DATA_BLOCK "dbVizu"
{ S7_Optimized_Access := 'FALSE' }
VERSION : 0.1
NON_RETAIN
   STRUCT
      iSecond : Int;
      iWMU_Temp : Int;   // 0,1°C
      iWMU_Ticks : Int;   // dílky   #0.1#°C#
      diAH1_Weight : DInt;   // 1g
      diAK1_Weight : DInt;   // 1g
      diAK2_Weight : DInt;   // 1g
      iAH1_TempSide : Int;   // 0,1°C
      iAH1_TempBottom : Int;   // 0,1°C
      iAK1_TempSide : Int;   // 0,1°C
      iAK1_TempBottom : Int;   // 0,1°C
      iAK2_TempSide : Int;   // 0,1°C
      iAK2_TempBottom : Int;   // 0,1°C
      iPIG1_Pressure : Int;   // 0,01 Bar
      iAK1_Pressure : Int;   // 0,01 Bar
      iAK2_Pressure : Int;   // 0,01 Bar
      iAH1_RCP_No : Int;   // cislo RCP
      usiAH1_RCP_Status : Byte;   // stav
      usiAH1_RCP_Step : Byte;   // krok
      sAH1_RCP_Name : String[40];   // jmeno RCP
      diAH1_RCP_TotalAmount : DInt;   // 0,001 kg
      iAH1_RCP_Shower_Step : Int;
      iAH1_RCP_TA : Int;
      diAH1_RCP_Mixture_need : DInt;   // 0,001 kg
      diAH1_RCP_Mixture_done : DInt;   // 0,001 kg
      diAH1_RCP_Mixing1_need : DInt;   // 0,016666667 min
      diAH1_RCP_Mixing1_done : DInt;   // 0,016666667 min
      diAH1_RCP_ManComp1_need : DInt;   // 0,001 kg
      diAH1_RCP_ManComp1_done : DInt;   // 0,001 kg
      diAH1_RCP_Mixing2_need : DInt;   // 0,016666667 min
      diAH1_RCP_Mixing2_done : DInt;   // 0,016666667 min
      diAH1_RCP_AutComp1_need : DInt;   // 0,001 kg
      diAH1_RCP_AutComp1_done : DInt;   // 0,001 kg
      diAH1_RCP_Mixing3_done : DInt;   // 0,016666667 min
      diAH1_RCP_Mixing3_need : DInt;   // 0,016666667 min
      iAH1_RCP_Ferm1_Temp : Int;   // 0,1 °C
      diAH1_RCP_Ferment1_need : DInt;   // 0,00027777778 hr
      diAH1_RCP_Ferment1_done : DInt;   // 0,00027777778 hr
      diAH1_RCP_ManComp2_need : DInt;   // 0,001 kg
      diAH1_RCP_ManComp2_done : DInt;   // 0,001 kg
      diAH1_RCP_Mixing4_need : DInt;   // 0,016666667 min
      diAH1_RCP_Mixing4_done : DInt;   // 0,016666667 min
      diAH1_RCP_AutComp2_need : DInt;   // 0,001 kg
      diAH1_RCP_AutComp2_done : DInt;   // 0,001 kg
      diAH1_RCP_Mixing5_done : DInt;   // 0,016666667 min
      diAH1_RCP_Mixing5_need : DInt;   // 0,016666667 min
      iAH1_RCP_Ferm2_Temp : Int;   // 0,1 °C
      diAH1_RCP_Ferment2_need : DInt;   // 0,00027777778 hr
      diAH1_RCP_Ferment2_done : DInt;   // 0,00027777778 hr
      iAH1_RCP_Repump1_Step : DInt;
      diAH1_RCP_LastWater_saved : DInt;
      diAH1_RCP_LastWater_curr : DInt;
      iAH1_RCP_Repump2_Step : Int;
      iAH1_RCP_PIG_Step : Int;
      iAH1_RCP_Clean_Step : Int;
      usiAH1_RCP_Dest : Byte;
      iAH1_Agit_Fwd_On : Int;   // s
      iAH1_Agit_Fwd_Off : Int;   // s
      iAH1_Agit_Fwd_Speed : Int;   // Hz
      iAH1_Agit_Rev_On : Int;   // s
      iAH1_Agit_Rev_Off : Int;   // s
      iAH1_Agit_Rev_Speed : Int;   // Hz
      usiAH1_RCP_Shower_Icon : Byte;
      usiAH1_RCP_Filling_Icon : Byte;
      usiAH1_RCP_Mixing1_Icon : Byte;
      usiAH1_RCP_ManComp1_Icon : Byte;
      usiAH1_RCP_Mixing2_Icon : Byte;
      usiAH1_RCP_AutComp1_Icon : Byte;
      usiAH1_RCP_Mixing3_Icon : Byte;
      usiAH1_RCP_Heat1_Icon : Byte;
      usiAH1_RCP_Ferment1_Icon : Byte;
      usiAH1_RCP_ManComp2_Icon : Byte;
      usiAH1_RCP_Mixing4_Icon : Byte;
      usiAH1_RCP_AutComp2_Icon : Byte;
      usiAH1_RCP_Mixing5_Icon : Byte;
      usiAH1_RCP_Heat2_Icon : Byte;
      usiAH1_RCP_Ferment2_Icon : Byte;
      usiAH1_RCP_Repump1_Icon : Byte;
      usiAH1_RCP_LastWater_Icon : Byte;
      usiAH1_RCP_Mixing6_Icon : Byte;
      usiAH1_RCP_Repump2_Icon : Byte;
      usiAH1_RCP_Pig_Icon : Byte;
      usiAH1_RCP_Cleaning_Icon : Byte;
      iAK1_RCP_No : Int;   // cislo RCP
      usiAK1_RCP_Status : Byte;   // stav
      usiAK1_RCP_Step : Byte;   // krok
      sAK1_RCP_Name : String[40];   // jmeno RCP
      diAK1_RCP_TotalAmount : DInt;
      iAK1_RCP_Shower_Step : Int;
      diAK1_RCP_Mixture_need : DInt;
      diAK1_RCP_Mixture_done : DInt;
      iAK1_RCP_Cooling_Temp : Int;   // 0,1 °C
      diAK1_RCP_Cooling_need : DInt;
      diAK1_RCP_Cooling_done : DInt;
      diAK1_RCP_Storing_need : DInt;   // 0,00027777778 hr
      diAK1_RCP_Storing_done : DInt;   // 0,00027777778 hr
      iAK1_RCP_Storing_Temp : Int;
      iAK1_RCP_CleanStep : Int;
      diAK1_RCP_Age : DInt;   // 0,00027777778 hr
      diAK1_RCP_AgeReady : DInt;   // 0,00027777778 hr
      diAK1_RCP_AgeMax : DInt;   // 0,00027777778 hr
      diAK1_BarLength : DInt;
      usiAK1_RCP_ProdStatus : Byte;
      usiAK1_RCP_Showering_Icon : Byte;
      usiAK1_RCP_Filling_Icon : Byte;
      usiAK1_RCP_Cooling_Icon : Byte;
      usiAK1_RCP_Storage_Icon : Byte;
      usiAK1_RCP_Cleaning_Icon : Byte;
      iAK1_Agit_Fwd_On : Int;   // s
      iAK1_Agit_Fwd_Off : Int;   // s
      iAK1_Agit_Rev_On : Int;   // s
      iAK1_Agit_Rev_Off : Int;   // s
      iAK1_ProdStatus : Int;
      iAK2_RCP_No : Int;   // cislo RCP
      usiAK2_RCP_Status : Byte;   // stav
      usiAK2_RCP_Step : Byte;   // krok
      sAK2_RCP_Name : String[40];   // jmeno RCP
      diAK2_RCP_TotalAmount : DInt;
      iAK2_RCP_Shower_Step : Int;
      diAK2_RCP_Mixture_need : DInt;
      diAK2_RCP_Mixture_done : DInt;
      iAK2_RCP_Cooling_Temp : Int;   // 0,1 °C
      diAK2_RCP_Cooling_need : DInt;
      diAK2_RCP_Cooling_done : DInt;
      diAK2_RCP_Storing_need : DInt;   // 0,00027777778 hr
      diAK2_RCP_Storing_done : DInt;   // 0,00027777778 hr
      iAK2_RCP_Storing_Temp : Int;
      iAK2_RCP_CleanStep : Int;
      diAK2_RCP_Age : DInt;   // 0,00027777778 hr
      diAK2_RCP_AgeReady : DInt;   // 0,00027777778 hr
      diAK2_RCP_AgeMax : DInt;   // 0,00027777778 hr
      diAK2_BarLength : DInt;
      usiAK2_RCP_ProdStatus : Byte;
      usiAK2_RCP_Showering_Icon : Byte;
      usiAK2_RCP_Filling_Icon : Byte;
      usiAK2_RCP_Cooling_Icon : Byte;
      usiAK2_RCP_Storage_Icon : Byte;
      usiAK2_RCP_Cleaning_Icon : Byte;
      iAK2_Agit_Fwd_On : Int;   // s
      iAK2_Agit_Fwd_Off : Int;   // s
      iAK2_Agit_Rev_On : Int;   // s
      iAK2_Agit_Rev_Off : Int;   // s
      iAK2_ProdStatus : Int;
      usiCleanTankAut_Status : Byte;
      usiCleanTankAut_Step : Byte;
      usiCleanTankAut_TankId : Byte;
      usiCleanTankAut_Owner : Byte;
      usiCleanTankMan_Status : Byte;
      usiCleanTankMan_Step : Byte;
      usiCleanTankMan_TankId : Byte;
      usiCleanTankMan_Owner : Byte;
      usiCleanTankWater_Status : Byte;
      usiCleanTankWater_Step : Byte;
      usiCleanTankWater_TankId : Byte;
      usiCleanTankWater_Owner : Byte;
      usiCleanTankShower_Status : Byte;
      usiCleanTankShower_Step : Byte;
      usiCleanTankShower_TankId : Byte;
      usiCleanTankShower_Owner : Byte;
      usiDischTank_Status : Byte;
      usiDischTank_Step : Byte;
      usiDischTank_TankId : Byte;
      usiDischTank_Owner : Byte;
      usiCleanPipe1_Status : Byte;
      usiCleanPipe1_Step : Byte;
      usiCleanPipe1_Owner : Byte;
      usiCleanPipe_Pig_1stStep : Byte;
      usiCleanPipe_Pig_2ndStep : Byte;
      usiPig1_Status : Byte;
      usiPig1_Step : Byte;
      usiPig1_LastPos : Byte;
      iPig1_LastDir : Int;
      usiPig1_Dest : Byte;
      usiPig1_Owner : Byte;
      usiDO_SourceTank : Byte;
      usiDO_Status : Byte;
      usiDO_Owner : Byte;
      bAH1_RCP_AutoClean : Bool;
      bAK1_RCP_AutoClean : Bool;
      bAK2_RCP_AutoClean : Bool;
      bAH1_LidOpen : Bool;
      bAK1_LidOpen : Bool;
      bAK2_LidOpen : Bool;
      bAH1_RepumAuto : Bool;
      bDO_AutoSelect : Bool;
      iEnd : Int;
   END_STRUCT;


BEGIN

END_DATA_BLOCK

